INTERFACE I_MotionDrive

PROPERTY CustomErrorMessage : STRING
GET
END_GET
SET
END_SET
END_PROPERTY

METHOD DepsInit
VAR_INPUT
END_VAR
END_METHOD

PROPERTY Done : BOOL
GET
END_GET
SET
END_SET
END_PROPERTY

PROPERTY Error : BOOL
GET
END_GET
SET
END_SET
END_PROPERTY

PROPERTY ErrorID : UDINT
GET
END_GET
SET
END_SET
END_PROPERTY

METHOD HandleInterFBCom
VAR_INPUT
END_VAR
END_METHOD

PROPERTY Name : STRING
GET
END_GET
SET
END_SET
END_PROPERTY

PROPERTY NegGoal : BOOL
GET
END_GET
SET
END_SET
END_PROPERTY

PROPERTY PosGoal : BOOL
GET
END_GET
SET
END_SET
END_PROPERTY

METHOD ProcessMoveReq
VAR_INPUT
END_VAR
END_METHOD

END_INTERFACE

(* stored: Version 1.1.0.1
   Itf I_MotionDrive: Id {4f84f724-7938-4847-ac53-18866323f75e}
   Property CustomErrorMessage: Id {1f202727-1b36-4e25-b74c-103d33b9d571}
   Get Get: Id {f8e06972-f73d-4bc3-9676-e2259d72e3ee}
   Set Set: Id {aae53a41-e997-4a33-a47e-083bd72a85ca}
   Method DepsInit: Id {bf5827d1-d917-4cf2-bee1-86b0b5256fcf}
   Property Done: Id {3f8a8de7-7e6f-415e-90b3-ae5922bd3074}
   Get Get: Id {e0481405-1904-426f-8294-683a0a15ba2c}
   Set Set: Id {69ec95aa-0883-4c80-92a1-83f7f5d53e54}
   Property Error: Id {28692bda-2e15-49a9-ae9c-44ee2c225402}
   Get Get: Id {e7c06eb5-1986-4004-bdcb-ca18cd302e3f}
   Set Set: Id {5320cbe2-83f6-49ab-a814-bb332a3d0b75}
   Property ErrorID: Id {415dcb0a-1a80-4f20-a5f6-d07b913efdcb}
   Get Get: Id {2080dd72-b57e-4aae-b589-16fc55f2d7f8}
   Set Set: Id {eb8abf2e-d9e9-4d6c-a6ee-9a201b51f0c5}
   Method HandleInterFBCom: Id {9db29681-ab2b-481a-8dad-3e40513073e7}
   Property Name: Id {808bc845-b6e4-4963-ab8f-244d15a3cc40}
   Get Get: Id {eef700d5-67cb-4093-abd3-49b2850feb0c}
   Set Set: Id {a8ad97b6-7dbe-4ad8-a2ac-9e24c41ccebb}
   Property NegGoal: Id {8ca9aaff-70e5-4a7d-a380-f334afbad2d7}
   Get Get: Id {dcb0f332-0cee-463b-a760-dfbb09a2481f}
   Set Set: Id {b6d4edb5-1521-4c30-ad4f-617130ebe079}
   Property PosGoal: Id {3bbc2f55-6d26-4fcf-84a1-58d794d496f9}
   Get Get: Id {c16d3cd5-bc57-4e01-b657-b628634e13d4}
   Set Set: Id {ab4cb165-b4bb-475f-901a-3072d677c7cc}
   Method ProcessMoveReq: Id {16636825-34ac-44bb-b4de-2566f4d18b17} *)
